// TIA Portal V19 export
FUNCTION "TEST_O_OUT_Fun" : Void   // FC205, LAD
// stored: SetENOAutomatically false
   VAR_TEMP   // added for the SCL form of the ladder/FBD networks
      _w1 : Bool;
   END_VAR
BEGIN

REGION Network 1
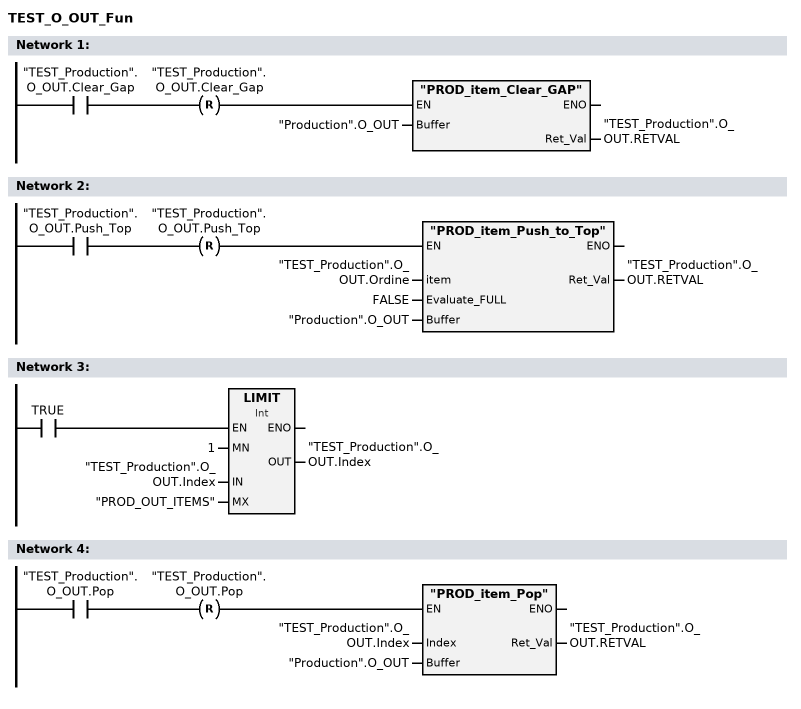
   RUNG wire#powerrail
      Contact( "TEST_Production".O_OUT.Clear_Gap )
      R_Coil( "TEST_Production".O_OUT.Clear_Gap )
      "PROD_item_Clear_GAP"(Buffer := "Production".O_OUT, Ret_Val => "TEST_Production".O_OUT.RETVAL)
   END_RUNG
   // the same network as SCL:
   #_w1 := "TEST_Production".O_OUT.Clear_Gap;
   IF #_w1 THEN
       "TEST_Production".O_OUT.Clear_Gap := FALSE;
       "TEST_Production".O_OUT.RETVAL := "PROD_item_Clear_GAP"(Buffer := "Production".O_OUT);
   END_IF;
END_REGION

REGION Network 2
   RUNG wire#powerrail
      Contact( "TEST_Production".O_OUT.Push_Top )
      R_Coil( "TEST_Production".O_OUT.Push_Top )
      "PROD_item_Push_to_Top"(item := "TEST_Production".O_OUT.Ordine, Evaluate_FULL := FALSE, Buffer := "Production".O_OUT, Ret_Val => "TEST_Production".O_OUT.RETVAL)
   END_RUNG
   // the same network as SCL:
   #_w1 := "TEST_Production".O_OUT.Push_Top;
   IF #_w1 THEN
       "TEST_Production".O_OUT.Push_Top := FALSE;
       "TEST_Production".O_OUT.RETVAL := "PROD_item_Push_to_Top"(item := "TEST_Production".O_OUT.Ordine,
                               Evaluate_FULL := FALSE,
                               Buffer := "Production".O_OUT);
   END_IF;
END_REGION

REGION Network 3
   RUNG wire#powerrail
      Contact( TRUE )
      { S7_Templates := "value_type := Int" } Limit(mn := 1, in := "TEST_Production".O_OUT.Index, mx := "PROD_OUT_ITEMS", out => "TEST_Production".O_OUT.Index)
   END_RUNG
   // the same network as SCL:
   IF TRUE THEN
       "TEST_Production".O_OUT.Index := LIMIT(MN := 1, IN := "TEST_Production".O_OUT.Index, MX := "PROD_OUT_ITEMS");
   END_IF;
END_REGION

REGION Network 4
   RUNG wire#powerrail
      Contact( "TEST_Production".O_OUT.Pop )
      R_Coil( "TEST_Production".O_OUT.Pop )
      "PROD_item_Pop"(Index := "TEST_Production".O_OUT.Index, Buffer := "Production".O_OUT, Ret_Val => "TEST_Production".O_OUT.RETVAL)
   END_RUNG
   // the same network as SCL:
   #_w1 := "TEST_Production".O_OUT.Pop;
   IF #_w1 THEN
       "TEST_Production".O_OUT.Pop := FALSE;
       "TEST_Production".O_OUT.RETVAL := "PROD_item_Pop"(Index := "TEST_Production".O_OUT.Index,
                               Buffer := "Production".O_OUT);
   END_IF;
END_REGION
END_FUNCTION
